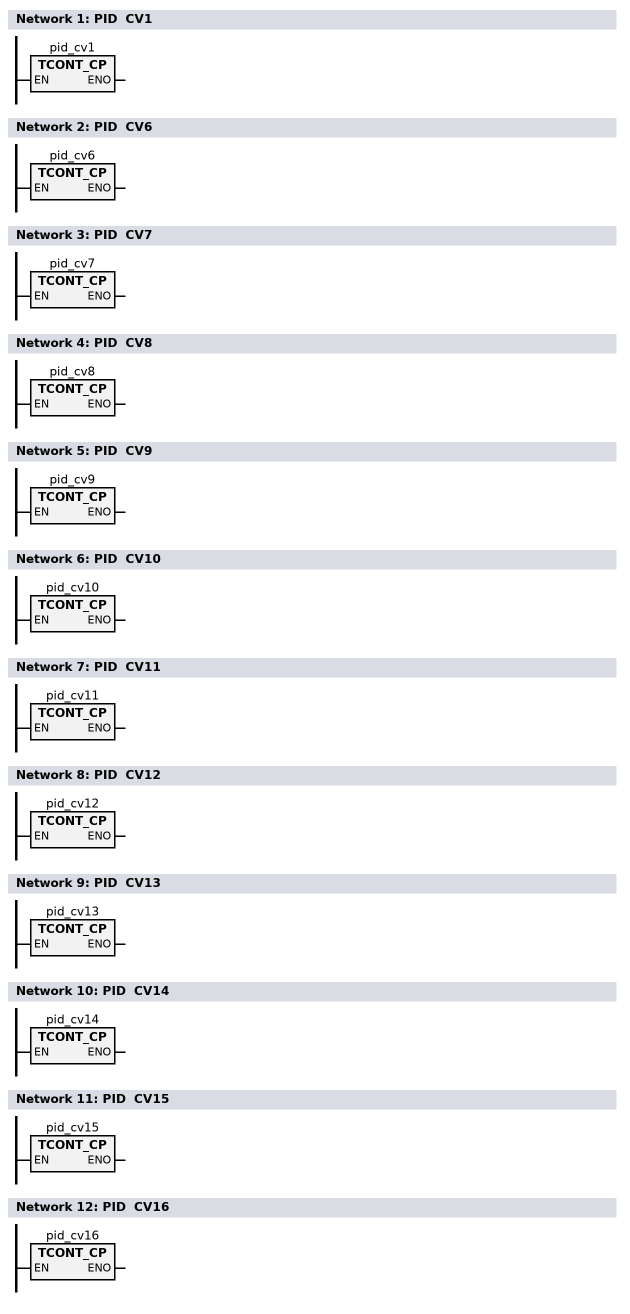
[picture p24: CYC_INT5 networks 1-12]
NETWORK
TITLE = PID  CV1
      CALL  "TCONT_CP" , "pid_cv1";
      NOP   0;
NETWORK
TITLE = PID  CV6
      CALL  "TCONT_CP" , "pid_cv6";
      NOP   0;
NETWORK
TITLE = PID  CV7
      CALL  "TCONT_CP" , "pid_cv7";
      NOP   0;
NETWORK
TITLE = PID  CV8
      CALL  "TCONT_CP" , "pid_cv8";
      NOP   0;
NETWORK
TITLE = PID  CV9
      CALL  "TCONT_CP" , "pid_cv9";
      NOP   0;
NETWORK
TITLE = PID  CV10
      CALL  "TCONT_CP" , "pid_cv10";
      NOP   0;
NETWORK
TITLE = PID  CV11
      CALL  "TCONT_CP" , "pid_cv11";
      NOP   0;
NETWORK
TITLE = PID  CV12
      CALL  "TCONT_CP" , "pid_cv12";
      NOP   0;
NETWORK
TITLE = PID  CV13
      CALL  "TCONT_CP" , "pid_cv13";
      NOP   0;
NETWORK
TITLE = PID  CV14
      CALL  "TCONT_CP" , "pid_cv14";
      NOP   0;
NETWORK
TITLE = PID  CV15
      CALL  "TCONT_CP" , "pid_cv15";
      NOP   0;
NETWORK
TITLE = PID  CV16
      CALL  "TCONT_CP" , "pid_cv16";
      NOP   0;
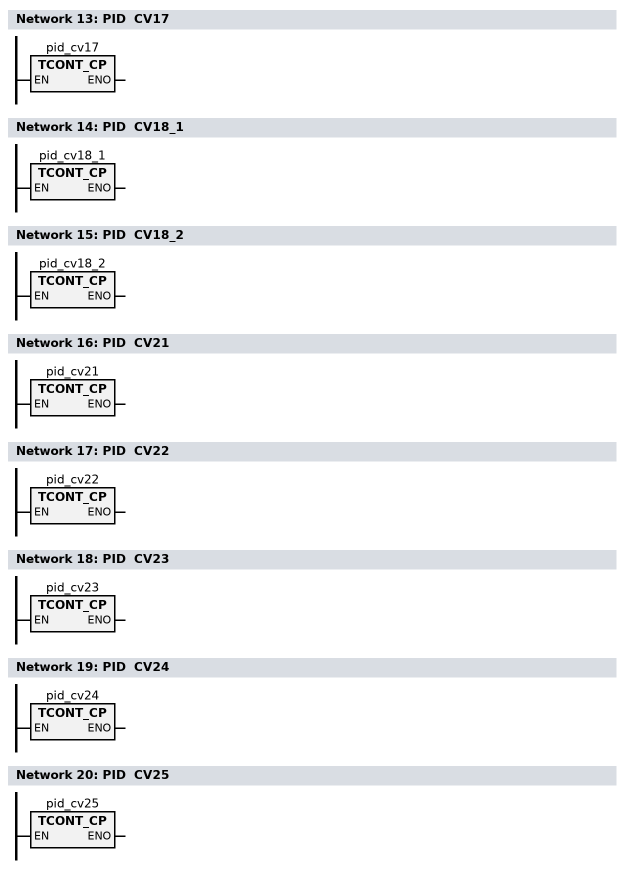
NETWORK
TITLE = PID  CV17
      CALL  "TCONT_CP" , "pid_cv17";
      NOP   0;
NETWORK
TITLE = PID  CV18_1
      CALL  "TCONT_CP" , "pid_cv18_1";
      NOP   0;
NETWORK
TITLE = PID  CV18_2
      CALL  "TCONT_CP" , "pid_cv18_2";
      NOP   0;
NETWORK
TITLE = PID  CV21
      CALL  "TCONT_CP" , "pid_cv21";
      NOP   0;
NETWORK
TITLE = PID  CV22
      CALL  "TCONT_CP" , "pid_cv22";
      NOP   0;
NETWORK
TITLE = PID  CV23
      CALL  "TCONT_CP" , "pid_cv23";
      NOP   0;
NETWORK
TITLE = PID  CV24
      CALL  "TCONT_CP" , "pid_cv24";
      NOP   0;
NETWORK
TITLE = PID  CV25
      CALL  "TCONT_CP" , "pid_cv25";
      NOP   0;
END_ORGANIZATION_BLOCK
